(* CoDeSys 2.3 export: ST_MODBUSADDRESSRANGE.EXP *)

(* Data type *)
TYPE ST_ModbusAddressRange :
STRUCT
	start: UINT;
	length: UINT;
	accessFunction: E_ModbusFunction;
END_STRUCT
END_TYPE
